ABB RobotStudio station: Path Planning V5 trial.rspag

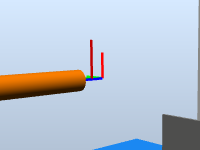
--- station ---
Station Path Planning V5 trial (saved by RobotStudio 6.8.8148.134)
Controller System310, task T_ROB1: task frame (RAPID world) sits at (0, 0, 305) mm in the station
Controller System310
  mechanical unit ROB_1: IRB2600_12_165_C_01, 6 joints, base frame (0, 0, 0) mm
Layout (positions relative to the parent item):
  - Bed [part, from Geometry\Bed.rslib]
  - Nozzle Support [part, from Geometry\Nozzle Support.rslib] at (138.01, 842.67, 817.43) mm, rotated rx -0.73 ry -0.25 rz 45.61 deg
  - Substrate Support [part, from Geometry\Substrate Support.rslib] at (485.68, 958.8, 1236.01) mm, rotated rx -0.25 ry 0.73 rz 135.61 deg
  - Table [part, from Geometry\Table.rslib] at (400.79, 567.93, 822.2) mm, rotated rx -0.73 ry -0.25 rz 45.61 deg
  - IRB2600_12_165_C_01 [mechanism, from Robots\IRB2600_12_165_C_01.rslib] at (0, 0, 305) mm; joint values [1.103, 0.1868, 0.1028, -0.014, 1.2809, 0.3109] (rad or m)
  - substrate_3 [part] at (499.49, 942.27, 926.24) mm, rotated rx -108.89 ry -89.23 rz 154.5 deg
Attachment: Substrate Support is attached to IRB2600_12_165_C_01 / Link6
Attachment: substrate_3 is attached to Substrate Support

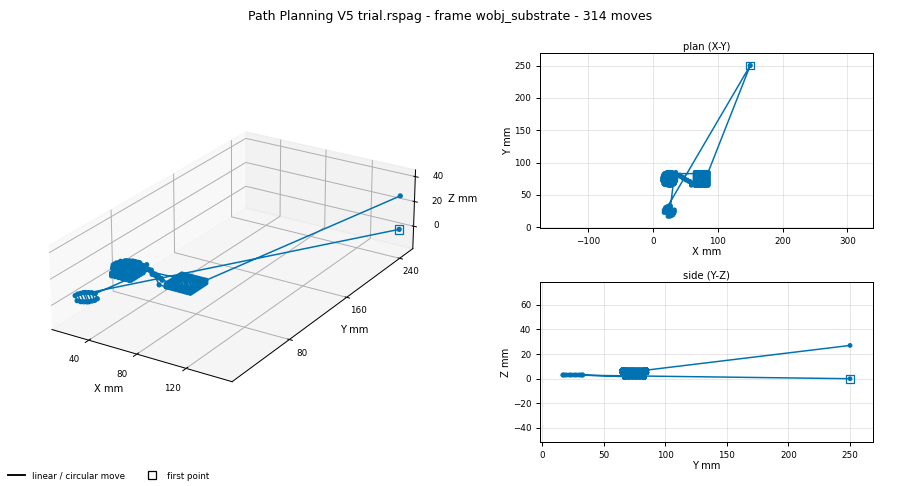
[picture p0: tool path of Path Planning V5 trial.rspag in frame wobj_substrate, 314 of 314 moves have a stored position in this frame; points joined in program order, loops and branches not executed]
--- Backups/System310/RAPID/TASK1/PROGMOD/MainModule.mod ---
MODULE MainModule
    TASK PERS tooldata tool_nozzle:=[FALSE,[[296.65274203,1095.137834363,767.916319098],[0.648657018,0.270531703,-0.654969146,0.277618601]],[1,[0,0,1],[1,0,0,0],0,0,0]];
    TASK PERS wobjdata wobj_substrate:=[TRUE,TRUE,"",[[8.5,-17.5,310],[0.707106781,0,0.707106781,0]],[[0,0,0],[1,0,0,0]]];

    VAR robtarget StartPoint:=[[150,250,0],[1,0,0,0],[-2,0,0,0],[9E+09,9E+09,9E+09,9E+09,9E+09,9E+09]];
    VAR robtarget ReferencePoint:=[[0,0,0],[1,0,0,0],[-2,0,0,0],[9E+09,9E+09,9E+09,9E+09,9E+09,9E+09]];
    VAR speeddata velocity_infill:=[90,500,5000,1000];
    VAR speeddata velocity_edge:=[45,500,5000,1000];
    VAR speeddata velocity_link:=[100,500,5000,1000];
    VAR zonedata zone_infill:=[FALSE,1,1,1,0.1,1,0.1];
    VAR zonedata zone_edge:=[FALSE,0.3,0.3,0.3,0.03,0.3,0.03];
    VAR zonedata zone_link:=[FALSE,5,8,8,0.8,8,0.8];

    PROC main()
        ConfJ\off;
        ConfL\Off;
        WaitTime 1;
        mod20260608;
    ENDPROC

    PROC mod20260608()
        MoveJ StartPoint,v100,fine,tool_nozzle\WObj:=wobj_substrate;
        MoveL RelTool(ReferencePoint,17,23,3\Rx:=0\Ry:=0\Rz:=0),velocity_infill,zone_infill,tool_nozzle\WObj:=wobj_substrate;
        MoveL RelTool(ReferencePoint,23,17,3\Rx:=0\Ry:=0\Rz:=0),velocity_infill,zone_infill,tool_nozzle\WObj:=wobj_substrate;
        MoveL RelTool(ReferencePoint,26,17,3\Rx:=0\Ry:=0\Rz:=0),velocity_infill,zone_infill,tool_nozzle\WObj:=wobj_substrate;
        MoveL RelTool(ReferencePoint,17,26,3\Rx:=0\Ry:=0\Rz:=0),velocity_infill,zone_infill,tool_nozzle\WObj:=wobj_substrate;
        MoveL RelTool(ReferencePoint,18,28,3\Rx:=0\Ry:=0\Rz:=0),velocity_infill,zone_infill,tool_nozzle\WObj:=wobj_substrate;
        MoveL RelTool(ReferencePoint,28,18,3\Rx:=0\Ry:=0\Rz:=0),velocity_infill,zone_infill,tool_nozzle\WObj:=wobj_substrate;
        MoveL RelTool(ReferencePoint,30,19,3\Rx:=0\Ry:=0\Rz:=0),velocity_infill,zone_infill,tool_nozzle\WObj:=wobj_substrate;
        MoveL RelTool(ReferencePoint,19,30,3\Rx:=0\Ry:=0\Rz:=0),velocity_infill,zone_infill,tool_nozzle\WObj:=wobj_substrate;
        MoveL RelTool(ReferencePoint,20,31,3\Rx:=0\Ry:=0\Rz:=0),velocity_infill,zone_infill,tool_nozzle\WObj:=wobj_substrate;
        MoveL RelTool(ReferencePoint,31,20,3\Rx:=0\Ry:=0\Rz:=0),velocity_infill,zone_infill,tool_nozzle\WObj:=wobj_substrate;
        MoveL RelTool(ReferencePoint,32,22,3\Rx:=0\Ry:=0\Rz:=0),velocity_infill,zone_infill,tool_nozzle\WObj:=wobj_substrate;
        MoveL RelTool(ReferencePoint,22,32,3\Rx:=0\Ry:=0\Rz:=0),velocity_infill,zone_infill,tool_nozzle\WObj:=wobj_substrate;
        MoveL RelTool(ReferencePoint,24,33,3\Rx:=0\Ry:=0\Rz:=0),velocity_infill,zone_infill,tool_nozzle\WObj:=wobj_substrate;
        MoveL RelTool(ReferencePoint,33,24,3\Rx:=0\Ry:=0\Rz:=0),velocity_infill,zone_infill,tool_nozzle\WObj:=wobj_substrate;
        MoveL RelTool(ReferencePoint,33,27,3\Rx:=0\Ry:=0\Rz:=0),velocity_infill,zone_infill,tool_nozzle\WObj:=wobj_substrate;
        MoveL RelTool(ReferencePoint,27,33,3\Rx:=0\Ry:=0\Rz:=0),velocity_infill,zone_infill,tool_nozzle\WObj:=wobj_substrate;
        MoveL RelTool(ReferencePoint,33,83,1\Rx:=0\Ry:=0\Rz:=0),velocity_infill,zone_infill,tool_nozzle\WObj:=wobj_substrate;
        MoveL RelTool(ReferencePoint,33,83,1\Rx:=0\Ry:=0\Rz:=0),velocity_infill,zone_infill,tool_nozzle\WObj:=wobj_substrate;
        MoveL RelTool(ReferencePoint,33,80,1\Rx:=0\Ry:=0\Rz:=0),velocity_infill,zone_infill,tool_nozzle\WObj:=wobj_substrate;
        MoveL RelTool(ReferencePoint,30,83,1\Rx:=0\Ry:=0\Rz:=0),velocity_infill,zone_infill,tool_nozzle\WObj:=wobj_substrate;
        MoveL RelTool(ReferencePoint,27,83,1\Rx:=0\Ry:=0\Rz:=0),velocity_infill,zone_infill,tool_nozzle\WObj:=wobj_substrate;
        MoveL RelTool(ReferencePoint,33,77,1\Rx:=0\Ry:=0\Rz:=0),velocity_infill,zone_infill,tool_nozzle\WObj:=wobj_substrate;
        MoveL RelTool(ReferencePoint,33,74,1\Rx:=0\Ry:=0\Rz:=0),velocity_infill,zone_infill,tool_nozzle\WObj:=wobj_substrate;
        MoveL RelTool(ReferencePoint,24,83,1\Rx:=0\Ry:=0\Rz:=0),velocity_infill,zone_infill,tool_nozzle\WObj:=wobj_substrate;
        MoveL RelTool(ReferencePoint,21,83,1\Rx:=0\Ry:=0\Rz:=0),velocity_infill,zone_infill,tool_nozzle\WObj:=wobj_substrate;
        MoveL RelTool(ReferencePoint,33,71,1\Rx:=0\Ry:=0\Rz:=0),velocity_infill,zone_infill,tool_nozzle\WObj:=wobj_substrate;
        MoveL RelTool(ReferencePoint,33,68,1\Rx:=0\Ry:=0\Rz:=0),velocity_infill,zone_infill,tool_nozzle\WObj:=wobj_substrate;
        MoveL RelTool(ReferencePoint,18,83,1\Rx:=0\Ry:=0\Rz:=0),velocity_infill,zone_infill,tool_nozzle\WObj:=wobj_substrate;
        MoveL RelTool(ReferencePoint,17,82,1\Rx:=0\Ry:=0\Rz:=0),velocity_infill,zone_infill,tool_nozzle\WObj:=wobj_substrate;
        MoveL RelTool(ReferencePoint,32,67,1\Rx:=0\Ry:=0\Rz:=0),velocity_infill,zone_infill,tool_nozzle\WObj:=wobj_substrate;
        MoveL RelTool(ReferencePoint,29,67,1\Rx:=0\Ry:=0\Rz:=0),velocity_infill,zone_infill,tool_nozzle\WObj:=wobj_substrate;
        MoveL RelTool(ReferencePoint,17,79,1\Rx:=0\Ry:=0\Rz:=0),velocity_infill,zone_infill,tool_nozzle\WObj:=wobj_substrate;
        MoveL RelTool(ReferencePoint,17,76,1\Rx:=0\Ry:=0\Rz:=0),velocity_infill,zone_infill,tool_nozzle\WObj:=wobj_substrate;
        MoveL RelTool(ReferencePoint,26,67,1\Rx:=0\Ry:=0\Rz:=0),velocity_infill,zone_infill,tool_nozzle\WObj:=wobj_substrate;
        MoveL RelTool(ReferencePoint,23,67,1\Rx:=0\Ry:=0\Rz:=0),velocity_infill,zone_infill,tool_nozzle\WObj:=wobj_substrate;
        MoveL RelTool(ReferencePoint,17,73,1\Rx:=0\Ry:=0\Rz:=0),velocity_infill,zone_infill,tool_nozzle\WObj:=wobj_substrate;
        MoveL RelTool(ReferencePoint,17,70,1\Rx:=0\Ry:=0\Rz:=0),velocity_infill,zone_infill,tool_nozzle\WObj:=wobj_substrate;
        MoveL RelTool(ReferencePoint,20,67,1\Rx:=0\Ry:=0\Rz:=0),velocity_infill,zone_infill,tool_nozzle\WObj:=wobj_substrate;
        MoveL RelTool(ReferencePoint,17,67,1\Rx:=0\Ry:=0\Rz:=0),velocity_infill,zone_infill,tool_nozzle\WObj:=wobj_substrate;
        MoveL RelTool(ReferencePoint,17,67,1\Rx:=0\Ry:=0\Rz:=0),velocity_infill,zone_infill,tool_nozzle\WObj:=wobj_substrate;
        MoveL RelTool(ReferencePoint,17,67,3\Rx:=0\Ry:=0\Rz:=0),velocity_infill,zone_infill,tool_nozzle\WObj:=wobj_substrate;
        MoveL RelTool(ReferencePoint,17,67,3\Rx:=0\Ry:=0\Rz:=0),velocity_infill,zone_infill,tool_nozzle\WObj:=wobj_substrate;
        MoveL RelTool(ReferencePoint,20,67,3\Rx:=0\Ry:=0\Rz:=0),velocity_infill,zone_infill,tool_nozzle\WObj:=wobj_substrate;
        MoveL RelTool(ReferencePoint,17,70,3\Rx:=0\Ry:=0\Rz:=0),velocity_infill,zone_infill,tool_nozzle\WObj:=wobj_substrate;
        MoveL RelTool(ReferencePoint,17,73,3\Rx:=0\Ry:=0\Rz:=0),velocity_infill,zone_infill,tool_nozzle\WObj:=wobj_substrate;
        MoveL RelTool(ReferencePoint,23,67,3\Rx:=0\Ry:=0\Rz:=0),velocity_infill,zone_infill,tool_nozzle\WObj:=wobj_substrate;
        MoveL RelTool(ReferencePoint,26,67,3\Rx:=0\Ry:=0\Rz:=0),velocity_infill,zone_infill,tool_nozzle\WObj:=wobj_substrate;
        MoveL RelTool(ReferencePoint,17,76,3\Rx:=0\Ry:=0\Rz:=0),velocity_infill,zone_infill,tool_nozzle\WObj:=wobj_substrate;
        MoveL RelTool(ReferencePoint,17,79,3\Rx:=0\Ry:=0\Rz:=0),velocity_infill,zone_infill,tool_nozzle\WObj:=wobj_substrate;
        MoveL RelTool(ReferencePoint,29,67,3\Rx:=0\Ry:=0\Rz:=0),velocity_infill,zone_infill,tool_nozzle\WObj:=wobj_substrate;
        MoveL RelTool(ReferencePoint,32,67,3\Rx:=0\Ry:=0\Rz:=0),velocity_infill,zone_infill,tool_nozzle\WObj:=wobj_substrate;
        MoveL RelTool(ReferencePoint,17,82,3\Rx:=0\Ry:=0\Rz:=0),velocity_infill,zone_infill,tool_nozzle\WObj:=wobj_substrate;
        MoveL RelTool(ReferencePoint,18,83,3\Rx:=0\Ry:=0\Rz:=0),velocity_infill,zone_infill,tool_nozzle\WObj:=wobj_substrate;
        MoveL RelTool(ReferencePoint,33,68,3\Rx:=0\Ry:=0\Rz:=0),velocity_infill,zone_infill,tool_nozzle\WObj:=wobj_substrate;
        MoveL RelTool(ReferencePoint,33,71,3\Rx:=0\Ry:=0\Rz:=0),velocity_infill,zone_infill,tool_nozzle\WObj:=wobj_substrate;
        MoveL RelTool(ReferencePoint,21,83,3\Rx:=0\Ry:=0\Rz:=0),velocity_infill,zone_infill,tool_nozzle\WObj:=wobj_substrate;
        MoveL RelTool(ReferencePoint,24,83,3\Rx:=0\Ry:=0\Rz:=0),velocity_infill,zone_infill,tool_nozzle\WObj:=wobj_substrate;
        MoveL RelTool(ReferencePoint,33,74,3\Rx:=0\Ry:=0\Rz:=0),velocity_infill,zone_infill,tool_nozzle\WObj:=wobj_substrate;
        MoveL RelTool(ReferencePoint,33,77,3\Rx:=0\Ry:=0\Rz:=0),velocity_infill,zone_infill,tool_nozzle\WObj:=wobj_substrate;
        MoveL RelTool(ReferencePoint,27,83,3\Rx:=0\Ry:=0\Rz:=0),velocity_infill,zone_infill,tool_nozzle\WObj:=wobj_substrate;
        MoveL RelTool(ReferencePoint,30,83,3\Rx:=0\Ry:=0\Rz:=0),velocity_infill,zone_infill,tool_nozzle\WObj:=wobj_substrate;
        MoveL RelTool(ReferencePoint,33,80,3\Rx:=0\Ry:=0\Rz:=0),velocity_infill,zone_infill,tool_nozzle\WObj:=wobj_substrate;
        MoveL RelTool(ReferencePoint,33,83,3\Rx:=0\Ry:=0\Rz:=0),velocity_infill,zone_infill,tool_nozzle\WObj:=wobj_substrate;
        MoveL RelTool(ReferencePoint,33,83,3\Rx:=0\Ry:=0\Rz:=0),velocity_infill,zone_infill,tool_nozzle\WObj:=wobj_substrate;
        MoveL RelTool(ReferencePoint,83,83,5\Rx:=0\Ry:=0\Rz:=0),velocity_infill,zone_infill,tool_nozzle\WObj:=wobj_substrate;
        MoveL RelTool(ReferencePoint,83,83,5\Rx:=0\Ry:=0\Rz:=0),velocity_infill,zone_infill,tool_nozzle\WObj:=wobj_substrate;
        MoveL RelTool(ReferencePoint,83,80,5\Rx:=0\Ry:=0\Rz:=0),velocity_infill,zone_infill,tool_nozzle\WObj:=wobj_substrate;
        MoveL RelTool(ReferencePoint,80,83,5\Rx:=0\Ry:=0\Rz:=0),velocity_infill,zone_infill,tool_nozzle\WObj:=wobj_substrate;
        MoveL RelTool(ReferencePoint,77,83,5\Rx:=0\Ry:=0\Rz:=0),velocity_infill,zone_infill,tool_nozzle\WObj:=wobj_substrate;
        MoveL RelTool(ReferencePoint,83,77,5\Rx:=0\Ry:=0\Rz:=0),velocity_infill,zone_infill,tool_nozzle\WObj:=wobj_substrate;
        MoveL RelTool(ReferencePoint,83,74,5\Rx:=0\Ry:=0\Rz:=0),velocity_infill,zone_infill,tool_nozzle\WObj:=wobj_substrate;
        MoveL RelTool(ReferencePoint,74,83,5\Rx:=0\Ry:=0\Rz:=0),velocity_infill,zone_infill,tool_nozzle\WObj:=wobj_substrate;
        MoveL RelTool(ReferencePoint,71,83,5\Rx:=0\Ry:=0\Rz:=0),velocity_infill,zone_infill,tool_nozzle\WObj:=wobj_substrate;
        MoveL RelTool(ReferencePoint,83,71,5\Rx:=0\Ry:=0\Rz:=0),velocity_infill,zone_infill,tool_nozzle\WObj:=wobj_substrate;
        MoveL RelTool(ReferencePoint,83,68,5\Rx:=0\Ry:=0\Rz:=0),velocity_infill,zone_infill,tool_nozzle\WObj:=wobj_substrate;
        MoveL RelTool(ReferencePoint,68,83,5\Rx:=0\Ry:=0\Rz:=0),velocity_infill,zone_infill,tool_nozzle\WObj:=wobj_substrate;
        MoveL RelTool(ReferencePoint,67,82,5\Rx:=0\Ry:=0\Rz:=0),velocity_infill,zone_infill,tool_nozzle\WObj:=wobj_substrate;
        MoveL RelTool(ReferencePoint,82,67,5\Rx:=0\Ry:=0\Rz:=0),velocity_infill,zone_infill,tool_nozzle\WObj:=wobj_substrate;
        MoveL RelTool(ReferencePoint,79,67,5\Rx:=0\Ry:=0\Rz:=0),velocity_infill,zone_infill,tool_nozzle\WObj:=wobj_substrate;
        MoveL RelTool(ReferencePoint,67,79,5\Rx:=0\Ry:=0\Rz:=0),velocity_infill,zone_infill,tool_nozzle\WObj:=wobj_substrate;
        MoveL RelTool(ReferencePoint,67,76,5\Rx:=0\Ry:=0\Rz:=0),velocity_infill,zone_infill,tool_nozzle\WObj:=wobj_substrate;
        MoveL RelTool(ReferencePoint,76,67,5\Rx:=0\Ry:=0\Rz:=0),velocity_infill,zone_infill,tool_nozzle\WObj:=wobj_substrate;
        MoveL RelTool(ReferencePoint,73,67,5\Rx:=0\Ry:=0\Rz:=0),velocity_infill,zone_infill,tool_nozzle\WObj:=wobj_substrate;
        MoveL RelTool(ReferencePoint,67,73,5\Rx:=0\Ry:=0\Rz:=0),velocity_infill,zone_infill,tool_nozzle\WObj:=wobj_substrate;
        MoveL RelTool(ReferencePoint,67,70,5\Rx:=0\Ry:=0\Rz:=0),velocity_infill,zone_infill,tool_nozzle\WObj:=wobj_substrate;
        MoveL RelTool(ReferencePoint,70,67,5\Rx:=0\Ry:=0\Rz:=0),velocity_infill,zone_infill,tool_nozzle\WObj:=wobj_substrate;
        MoveL RelTool(ReferencePoint,67,67,5\Rx:=0\Ry:=0\Rz:=0),velocity_infill,zone_infill,tool_nozzle\WObj:=wobj_substrate;
        MoveL RelTool(ReferencePoint,67,67,5\Rx:=0\Ry:=0\Rz:=0),velocity_infill,zone_infill,tool_nozzle\WObj:=wobj_substrate;
        MoveL RelTool(ReferencePoint,65,65,5\Rx:=0\Ry:=-30\Rz:=0),velocity_edge,zone_edge,tool_nozzle\WObj:=wobj_substrate;
        MoveL RelTool(ReferencePoint,65,67,5\Rx:=0\Ry:=-30\Rz:=0),velocity_edge,zone_edge,tool_nozzle\WObj:=wobj_substrate;
        MoveL RelTool(ReferencePoint,65,69,5\Rx:=0\Ry:=-30\Rz:=0),velocity_edge,zone_edge,tool_nozzle\WObj:=wobj_substrate;
        MoveL RelTool(ReferencePoint,65,71,5\Rx:=0\Ry:=-30\Rz:=0),velocity_edge,zone_edge,tool_nozzle\WObj:=wobj_substrate;
        MoveL RelTool(ReferencePoint,65,73,5\Rx:=0\Ry:=-30\Rz:=0),velocity_edge,zone_edge,tool_nozzle\WObj:=wobj_substrate;
        MoveL RelTool(ReferencePoint,65,75,5\Rx:=0\Ry:=-30\Rz:=0),velocity_edge,zone_edge,tool_nozzle\WObj:=wobj_substrate;
        MoveL RelTool(ReferencePoint,65,77,5\Rx:=0\Ry:=-30\Rz:=0),velocity_edge,zone_edge,tool_nozzle\WObj:=wobj_substrate;
        MoveL RelTool(ReferencePoint,65,79,5\Rx:=0\Ry:=-30\Rz:=0),velocity_edge,zone_edge,tool_nozzle\WObj:=wobj_substrate;
        MoveL RelTool(ReferencePoint,65,81,5\Rx:=0\Ry:=-30\Rz:=0),velocity_edge,zone_edge,tool_nozzle\WObj:=wobj_substrate;
        MoveL RelTool(ReferencePoint,65,83,5\Rx:=0\Ry:=-30\Rz:=0),velocity_edge,zone_edge,tool_nozzle\WObj:=wobj_substrate;
        MoveL RelTool(ReferencePoint,65,85,5\Rx:=-30\Ry:=0\Rz:=0),velocity_edge,zone_edge,tool_nozzle\WObj:=wobj_substrate;
        MoveL RelTool(ReferencePoint,67,85,5\Rx:=-30\Ry:=0\Rz:=0),velocity_edge,zone_edge,tool_nozzle\WObj:=wobj_substrate;
        MoveL RelTool(ReferencePoint,69,85,5\Rx:=-30\Ry:=0\Rz:=0),velocity_edge,zone_edge,tool_nozzle\WObj:=wobj_substrate;
        MoveL RelTool(ReferencePoint,71,85,5\Rx:=-30\Ry:=0\Rz:=0),velocity_edge,zone_edge,tool_nozzle\WObj:=wobj_substrate;
        MoveL RelTool(ReferencePoint,73,85,5\Rx:=-30\Ry:=0\Rz:=0),velocity_edge,zone_edge,tool_nozzle\WObj:=wobj_substrate;
        MoveL RelTool(ReferencePoint,75,85,5\Rx:=-30\Ry:=0\Rz:=0),velocity_edge,zone_edge,tool_nozzle\WObj:=wobj_substrate;
        MoveL RelTool(ReferencePoint,77,85,5\Rx:=-30\Ry:=0\Rz:=0),velocity_edge,zone_edge,tool_nozzle\WObj:=wobj_substrate;
        MoveL RelTool(ReferencePoint,79,85,5\Rx:=-30\Ry:=0\Rz:=0),velocity_edge,zone_edge,tool_nozzle\WObj:=wobj_substrate;
        MoveL RelTool(ReferencePoint,81,85,5\Rx:=-30\Ry:=0\Rz:=0),velocity_edge,zone_edge,tool_nozzle\WObj:=wobj_substrate;
        MoveL RelTool(ReferencePoint,83,85,5\Rx:=-30\Ry:=0\Rz:=0),velocity_edge,zone_edge,tool_nozzle\WObj:=wobj_substrate;
        MoveL RelTool(ReferencePoint,85,85,5\Rx:=0\Ry:=30\Rz:=0),velocity_edge,zone_edge,tool_nozzle\WObj:=wobj_substrate;
        MoveL RelTool(ReferencePoint,85,83,5\Rx:=0\Ry:=30\Rz:=0),velocity_edge,zone_edge,tool_nozzle\WObj:=wobj_substrate;
        MoveL RelTool(ReferencePoint,85,81,5\Rx:=0\Ry:=30\Rz:=0),velocity_edge,zone_edge,tool_nozzle\WObj:=wobj_substrate;
        MoveL RelTool(ReferencePoint,85,79,5\Rx:=0\Ry:=30\Rz:=0),velocity_edge,zone_edge,tool_nozzle\WObj:=wobj_substrate;
        MoveL RelTool(ReferencePoint,85,77,5\Rx:=0\Ry:=30\Rz:=0),velocity_edge,zone_edge,tool_nozzle\WObj:=wobj_substrate;
        MoveL RelTool(ReferencePoint,85,75,5\Rx:=0\Ry:=30\Rz:=0),velocity_edge,zone_edge,tool_nozzle\WObj:=wobj_substrate;
        MoveL RelTool(ReferencePoint,85,73,5\Rx:=0\Ry:=30\Rz:=0),velocity_edge,zone_edge,tool_nozzle\WObj:=wobj_substrate;
        MoveL RelTool(ReferencePoint,85,71,5\Rx:=0\Ry:=30\Rz:=0),velocity_edge,zone_edge,tool_nozzle\WObj:=wobj_substrate;
        MoveL RelTool(ReferencePoint,85,69,5\Rx:=0\Ry:=30\Rz:=0),velocity_edge,zone_edge,tool_nozzle\WObj:=wobj_substrate;
        MoveL RelTool(ReferencePoint,85,67,5\Rx:=0\Ry:=30\Rz:=0),velocity_edge,zone_edge,tool_nozzle\WObj:=wobj_substrate;
        MoveL RelTool(ReferencePoint,85,65,5\Rx:=30\Ry:=0\Rz:=0),velocity_edge,zone_edge,tool_nozzle\WObj:=wobj_substrate;
        MoveL RelTool(ReferencePoint,83,65,5\Rx:=30\Ry:=0\Rz:=0),velocity_edge,zone_edge,tool_nozzle\WObj:=wobj_substrate;
        MoveL RelTool(ReferencePoint,81,65,5\Rx:=30\Ry:=0\Rz:=0),velocity_edge,zone_edge,tool_nozzle\WObj:=wobj_substrate;
        MoveL RelTool(ReferencePoint,79,65,5\Rx:=30\Ry:=0\Rz:=0),velocity_edge,zone_edge,tool_nozzle\WObj:=wobj_substrate;
        MoveL RelTool(ReferencePoint,77,65,5\Rx:=30\Ry:=0\Rz:=0),velocity_edge,zone_edge,tool_nozzle\WObj:=wobj_substrate;
        MoveL RelTool(ReferencePoint,75,65,5\Rx:=30\Ry:=0\Rz:=0),velocity_edge,zone_edge,tool_nozzle\WObj:=wobj_substrate;
        MoveL RelTool(ReferencePoint,73,65,5\Rx:=30\Ry:=0\Rz:=0),velocity_edge,zone_edge,tool_nozzle\WObj:=wobj_substrate;
        MoveL RelTool(ReferencePoint,71,65,5\Rx:=30\Ry:=0\Rz:=0),velocity_edge,zone_edge,tool_nozzle\WObj:=wobj_substrate;
        MoveL RelTool(ReferencePoint,69,65,5\Rx:=30\Ry:=0\Rz:=0),velocity_edge,zone_edge,tool_nozzle\WObj:=wobj_substrate;
        MoveL RelTool(ReferencePoint,67,65,5\Rx:=30\Ry:=0\Rz:=0),velocity_edge,zone_edge,tool_nozzle\WObj:=wobj_substrate;
        MoveL RelTool(ReferencePoint,65,65,5\Rx:=30\Ry:=0\Rz:=0),velocity_edge,zone_edge,tool_nozzle\WObj:=wobj_substrate;
        MoveL RelTool(ReferencePoint,65,65,5\Rx:=0\Ry:=0\Rz:=0),velocity_link,zone_link,tool_nozzle\WObj:=wobj_substrate;
        MoveL RelTool(ReferencePoint,59,65,5\Rx:=0\Ry:=0\Rz:=0),velocity_link,zone_link,tool_nozzle\WObj:=wobj_substrate;
        MoveL RelTool(ReferencePoint,47,77,5\Rx:=0\Ry:=0\Rz:=0),velocity_link,zone_link,tool_nozzle\WObj:=wobj_substrate;
        MoveL RelTool(ReferencePoint,45,77,5\Rx:=0\Ry:=0\Rz:=0),velocity_link,zone_link,tool_nozzle\WObj:=wobj_substrate;
        MoveL RelTool(ReferencePoint,41,81,5\Rx:=0\Ry:=0\Rz:=0),velocity_link,zone_link,tool_nozzle\WObj:=wobj_substrate;
        MoveL RelTool(ReferencePoint,37,81,5\Rx:=0\Ry:=0\Rz:=0),velocity_link,zone_link,tool_nozzle\WObj:=wobj_substrate;
        MoveL RelTool(ReferencePoint,35,83,5\Rx:=0\Ry:=0\Rz:=0),velocity_link,zone_link,tool_nozzle\WObj:=wobj_substrate;
        MoveL RelTool(ReferencePoint,29,83,5\Rx:=0\Ry:=0\Rz:=0),velocity_link,zone_link,tool_nozzle\WObj:=wobj_substrate;
        MoveL RelTool(ReferencePoint,27,83,5\Rx:=0\Ry:=0\Rz:=0),velocity_infill,zone_infill,tool_nozzle\WObj:=wobj_substrate;
        MoveL RelTool(ReferencePoint,33,77,5\Rx:=0\Ry:=0\Rz:=0),velocity_infill,zone_infill,tool_nozzle\WObj:=wobj_substrate;
        MoveL RelTool(ReferencePoint,33,74,5\Rx:=0\Ry:=0\Rz:=0),velocity_infill,zone_infill,tool_nozzle\WObj:=wobj_substrate;
        MoveL RelTool(ReferencePoint,24,83,5\Rx:=0\Ry:=0\Rz:=0),velocity_infill,zone_infill,tool_nozzle\WObj:=wobj_substrate;
        MoveL RelTool(ReferencePoint,22,82,5\Rx:=0\Ry:=0\Rz:=0),velocity_infill,zone_infill,tool_nozzle\WObj:=wobj_substrate;
        MoveL RelTool(ReferencePoint,32,72,5\Rx:=0\Ry:=0\Rz:=0),velocity_infill,zone_infill,tool_nozzle\WObj:=wobj_substrate;
        MoveL RelTool(ReferencePoint,31,70,5\Rx:=0\Ry:=0\Rz:=0),velocity_infill,zone_infill,tool_nozzle\WObj:=wobj_substrate;
        MoveL RelTool(ReferencePoint,20,81,5\Rx:=0\Ry:=0\Rz:=0),velocity_infill,zone_infill,tool_nozzle\WObj:=wobj_substrate;
        MoveL RelTool(ReferencePoint,19,80,5\Rx:=0\Ry:=0\Rz:=0),velocity_infill,zone_infill,tool_nozzle\WObj:=wobj_substrate;
        MoveL RelTool(ReferencePoint,30,69,5\Rx:=0\Ry:=0\Rz:=0),velocity_infill,zone_infill,tool_nozzle\WObj:=wobj_substrate;
        MoveL RelTool(ReferencePoint,28,68,5\Rx:=0\Ry:=0\Rz:=0),velocity_infill,zone_infill,tool_nozzle\WObj:=wobj_substrate;
        MoveL RelTool(ReferencePoint,18,78,5\Rx:=0\Ry:=0\Rz:=0),velocity_infill,zone_infill,tool_nozzle\WObj:=wobj_substrate;
        MoveL RelTool(ReferencePoint,17,76,5\Rx:=0\Ry:=0\Rz:=0),velocity_infill,zone_infill,tool_nozzle\WObj:=wobj_substrate;
        MoveL RelTool(ReferencePoint,26,67,5\Rx:=0\Ry:=0\Rz:=0),velocity_infill,zone_infill,tool_nozzle\WObj:=wobj_substrate;
        MoveL RelTool(ReferencePoint,23,67,5\Rx:=0\Ry:=0\Rz:=0),velocity_infill,zone_infill,tool_nozzle\WObj:=wobj_substrate;
        MoveL RelTool(ReferencePoint,17,73,5\Rx:=0\Ry:=0\Rz:=0),velocity_infill,zone_infill,tool_nozzle\WObj:=wobj_substrate;
        MoveL RelTool(ReferencePoint,15,72,5\Rx:=8\Ry:=-29\Rz:=0),velocity_edge,zone_edge,tool_nozzle\WObj:=wobj_substrate;
        MoveL RelTool(ReferencePoint,15,74,5\Rx:=2\Ry:=-30\Rz:=0),velocity_edge,zone_edge,tool_nozzle\WObj:=wobj_substrate;
        MoveL RelTool(ReferencePoint,15,76,5\Rx:=-5\Ry:=-30\Rz:=0),velocity_edge,zone_edge,tool_nozzle\WObj:=wobj_substrate;
        MoveL RelTool(ReferencePoint,15,78,5\Rx:=-11\Ry:=-28\Rz:=0),velocity_edge,zone_edge,tool_nozzle\WObj:=wobj_substrate;
        MoveL RelTool(ReferencePoint,16,80,5\Rx:=-17\Ry:=-25\Rz:=0),velocity_edge,zone_edge,tool_nozzle\WObj:=wobj_substrate;
        MoveL RelTool(ReferencePoint,17,81,5\Rx:=-21\Ry:=-22\Rz:=0),velocity_edge,zone_edge,tool_nozzle\WObj:=wobj_substrate;
        MoveL RelTool(ReferencePoint,19,83,5\Rx:=-25\Ry:=-17\Rz:=0),velocity_edge,zone_edge,tool_nozzle\WObj:=wobj_substrate;
        MoveL RelTool(ReferencePoint,21,84,5\Rx:=-28\Ry:=-12\Rz:=0),velocity_edge,zone_edge,tool_nozzle\WObj:=wobj_substrate;
        MoveL RelTool(ReferencePoint,22,85,5\Rx:=-29\Ry:=-7\Rz:=0),velocity_edge,zone_edge,tool_nozzle\WObj:=wobj_substrate;
        MoveL RelTool(ReferencePoint,24,85,5\Rx:=-30\Ry:=-1\Rz:=0),velocity_edge,zone_edge,tool_nozzle\WObj:=wobj_substrate;
        MoveL RelTool(ReferencePoint,26,85,5\Rx:=-30\Ry:=4\Rz:=0),velocity_edge,zone_edge,tool_nozzle\WObj:=wobj_substrate;
        MoveL RelTool(ReferencePoint,28,84,5\Rx:=-29\Ry:=10\Rz:=0),velocity_edge,zone_edge,tool_nozzle\WObj:=wobj_substrate;
        MoveL RelTool(ReferencePoint,30,84,5\Rx:=-26\Ry:=15\Rz:=0),velocity_edge,zone_edge,tool_nozzle\WObj:=wobj_substrate;
        MoveL RelTool(ReferencePoint,32,82,5\Rx:=-23\Ry:=20\Rz:=0),velocity_edge,zone_edge,tool_nozzle\WObj:=wobj_substrate;
        MoveL RelTool(ReferencePoint,33,81,5\Rx:=-19\Ry:=24\Rz:=0),velocity_edge,zone_edge,tool_nozzle\WObj:=wobj_substrate;
        MoveL RelTool(ReferencePoint,34,79,5\Rx:=-14\Ry:=27\Rz:=0),velocity_edge,zone_edge,tool_nozzle\WObj:=wobj_substrate;
        MoveL RelTool(ReferencePoint,35,77,5\Rx:=-8\Ry:=29\Rz:=0),velocity_edge,zone_edge,tool_nozzle\WObj:=wobj_substrate;
        MoveL RelTool(ReferencePoint,35,75,5\Rx:=-2\Ry:=30\Rz:=0),velocity_edge,zone_edge,tool_nozzle\WObj:=wobj_substrate;
        MoveL RelTool(ReferencePoint,35,73,5\Rx:=5\Ry:=30\Rz:=0),velocity_edge,zone_edge,tool_nozzle\WObj:=wobj_substrate;
        MoveL RelTool(ReferencePoint,34,71,5\Rx:=11\Ry:=28\Rz:=0),velocity_edge,zone_edge,tool_nozzle\WObj:=wobj_substrate;
        MoveL RelTool(ReferencePoint,33,70,5\Rx:=17\Ry:=25\Rz:=0),velocity_edge,zone_edge,tool_nozzle\WObj:=wobj_substrate;
        MoveL RelTool(ReferencePoint,32,68,5\Rx:=21\Ry:=22\Rz:=0),velocity_edge,zone_edge,tool_nozzle\WObj:=wobj_substrate;
        MoveL RelTool(ReferencePoint,31,67,5\Rx:=25\Ry:=17\Rz:=0),velocity_edge,zone_edge,tool_nozzle\WObj:=wobj_substrate;
        MoveL RelTool(ReferencePoint,29,66,5\Rx:=28\Ry:=12\Rz:=0),velocity_edge,zone_edge,tool_nozzle\WObj:=wobj_substrate;
        MoveL RelTool(ReferencePoint,27,65,5\Rx:=29\Ry:=7\Rz:=0),velocity_edge,zone_edge,tool_nozzle\WObj:=wobj_substrate;
        MoveL RelTool(ReferencePoint,25,65,5\Rx:=30\Ry:=1\Rz:=0),velocity_edge,zone_edge,tool_nozzle\WObj:=wobj_substrate;
        MoveL RelTool(ReferencePoint,23,65,5\Rx:=30\Ry:=-4\Rz:=0),velocity_edge,zone_edge,tool_nozzle\WObj:=wobj_substrate;
        MoveL RelTool(ReferencePoint,21,66,5\Rx:=28\Ry:=-12\Rz:=0),velocity_edge,zone_edge,tool_nozzle\WObj:=wobj_substrate;
        MoveL RelTool(ReferencePoint,19,67,5\Rx:=25\Ry:=-17\Rz:=0),velocity_edge,zone_edge,tool_nozzle\WObj:=wobj_substrate;
        MoveL RelTool(ReferencePoint,18,68,5\Rx:=21\Ry:=-22\Rz:=0),velocity_edge,zone_edge,tool_nozzle\WObj:=wobj_substrate;
        MoveL RelTool(ReferencePoint,17,70,5\Rx:=17\Ry:=-25\Rz:=0),velocity_edge,zone_edge,tool_nozzle\WObj:=wobj_substrate;
        MoveL RelTool(ReferencePoint,16,71,5\Rx:=11\Ry:=-28\Rz:=0),velocity_edge,zone_edge,tool_nozzle\WObj:=wobj_substrate;
        MoveL RelTool(ReferencePoint,15,72,5\Rx:=9\Ry:=-29\Rz:=0),velocity_edge,zone_edge,tool_nozzle\WObj:=wobj_substrate;
        MoveL RelTool(ReferencePoint,17,73,7\Rx:=0\Ry:=0\Rz:=0),velocity_infill,zone_infill,tool_nozzle\WObj:=wobj_substrate;
        MoveL RelTool(ReferencePoint,23,67,7\Rx:=0\Ry:=0\Rz:=0),velocity_infill,zone_infill,tool_nozzle\WObj:=wobj_substrate;
        MoveL RelTool(ReferencePoint,26,67,7\Rx:=0\Ry:=0\Rz:=0),velocity_infill,zone_infill,tool_nozzle\WObj:=wobj_substrate;
        MoveL RelTool(ReferencePoint,17,76,7\Rx:=0\Ry:=0\Rz:=0),velocity_infill,zone_infill,tool_nozzle\WObj:=wobj_substrate;
        MoveL RelTool(ReferencePoint,18,78,7\Rx:=0\Ry:=0\Rz:=0),velocity_infill,zone_infill,tool_nozzle\WObj:=wobj_substrate;
        MoveL RelTool(ReferencePoint,28,68,7\Rx:=0\Ry:=0\Rz:=0),velocity_infill,zone_infill,tool_nozzle\WObj:=wobj_substrate;
        MoveL RelTool(ReferencePoint,30,69,7\Rx:=0\Ry:=0\Rz:=0),velocity_infill,zone_infill,tool_nozzle\WObj:=wobj_substrate;
        MoveL RelTool(ReferencePoint,19,80,7\Rx:=0\Ry:=0\Rz:=0),velocity_infill,zone_infill,tool_nozzle\WObj:=wobj_substrate;
        MoveL RelTool(ReferencePoint,20,81,7\Rx:=0\Ry:=0\Rz:=0),velocity_infill,zone_infill,tool_nozzle\WObj:=wobj_substrate;
        MoveL RelTool(ReferencePoint,31,70,7\Rx:=0\Ry:=0\Rz:=0),velocity_infill,zone_infill,tool_nozzle\WObj:=wobj_substrate;
        MoveL RelTool(ReferencePoint,32,72,7\Rx:=0\Ry:=0\Rz:=0),velocity_infill,zone_infill,tool_nozzle\WObj:=wobj_substrate;
        MoveL RelTool(ReferencePoint,22,82,7\Rx:=0\Ry:=0\Rz:=0),velocity_infill,zone_infill,tool_nozzle\WObj:=wobj_substrate;
        MoveL RelTool(ReferencePoint,24,83,7\Rx:=0\Ry:=0\Rz:=0),velocity_infill,zone_infill,tool_nozzle\WObj:=wobj_substrate;
        MoveL RelTool(ReferencePoint,33,74,7\Rx:=0\Ry:=0\Rz:=0),velocity_infill,zone_infill,tool_nozzle\WObj:=wobj_substrate;
        MoveL RelTool(ReferencePoint,33,77,7\Rx:=0\Ry:=0\Rz:=0),velocity_infill,zone_infill,tool_nozzle\WObj:=wobj_substrate;
        MoveL RelTool(ReferencePoint,27,83,7\Rx:=0\Ry:=0\Rz:=0),velocity_infill,zone_infill,tool_nozzle\WObj:=wobj_substrate;
        MoveL RelTool(ReferencePoint,28,85,7\Rx:=-29\Ry:=7\Rz:=0),velocity_edge,zone_edge,tool_nozzle\WObj:=wobj_substrate;
        MoveL RelTool(ReferencePoint,29,84,7\Rx:=-28\Ry:=12\Rz:=0),velocity_edge,zone_edge,tool_nozzle\WObj:=wobj_substrate;
        MoveL RelTool(ReferencePoint,31,83,7\Rx:=-24\Ry:=18\Rz:=0),velocity_edge,zone_edge,tool_nozzle\WObj:=wobj_substrate;
        MoveL RelTool(ReferencePoint,33,82,7\Rx:=-21\Ry:=22\Rz:=0),velocity_edge,zone_edge,tool_nozzle\WObj:=wobj_substrate;
        MoveL RelTool(ReferencePoint,34,80,7\Rx:=-15\Ry:=26\Rz:=0),velocity_edge,zone_edge,tool_nozzle\WObj:=wobj_substrate;
        MoveL RelTool(ReferencePoint,34,78,7\Rx:=-11\Ry:=28\Rz:=0),velocity_edge,zone_edge,tool_nozzle\WObj:=wobj_substrate;
        MoveL RelTool(ReferencePoint,35,76,7\Rx:=-2\Ry:=30\Rz:=0),velocity_edge,zone_edge,tool_nozzle\WObj:=wobj_substrate;
        MoveL RelTool(ReferencePoint,35,74,7\Rx:=2\Ry:=30\Rz:=0),velocity_edge,zone_edge,tool_nozzle\WObj:=wobj_substrate;
        MoveL RelTool(ReferencePoint,35,72,7\Rx:=8\Ry:=29\Rz:=0),velocity_edge,zone_edge,tool_nozzle\WObj:=wobj_substrate;
        MoveL RelTool(ReferencePoint,34,70,7\Rx:=15\Ry:=26\Rz:=0),velocity_edge,zone_edge,tool_nozzle\WObj:=wobj_substrate;
        MoveL RelTool(ReferencePoint,33,69,7\Rx:=19\Ry:=24\Rz:=0),velocity_edge,zone_edge,tool_nozzle\WObj:=wobj_substrate;
        MoveL RelTool(ReferencePoint,31,67,7\Rx:=24\Ry:=18\Rz:=0),velocity_edge,zone_edge,tool_nozzle\WObj:=wobj_substrate;
        MoveL RelTool(ReferencePoint,30,66,7\Rx:=27\Ry:=14\Rz:=0),velocity_edge,zone_edge,tool_nozzle\WObj:=wobj_substrate;
        MoveL RelTool(ReferencePoint,28,65,7\Rx:=29\Ry:=7\Rz:=0),velocity_edge,zone_edge,tool_nozzle\WObj:=wobj_substrate;
        MoveL RelTool(ReferencePoint,26,65,7\Rx:=30\Ry:=3\Rz:=0),velocity_edge,zone_edge,tool_nozzle\WObj:=wobj_substrate;
        MoveL RelTool(ReferencePoint,24,65,7\Rx:=30\Ry:=-4\Rz:=0),velocity_edge,zone_edge,tool_nozzle\WObj:=wobj_substrate;
        MoveL RelTool(ReferencePoint,22,66,7\Rx:=29\Ry:=-9\Rz:=0),velocity_edge,zone_edge,tool_nozzle\WObj:=wobj_substrate;
        MoveL RelTool(ReferencePoint,20,66,7\Rx:=26\Ry:=-15\Rz:=0),velocity_edge,zone_edge,tool_nozzle\WObj:=wobj_substrate;
        MoveL RelTool(ReferencePoint,18,67,7\Rx:=23\Ry:=-20\Rz:=0),velocity_edge,zone_edge,tool_nozzle\WObj:=wobj_substrate;
        MoveL RelTool(ReferencePoint,17,69,7\Rx:=19\Ry:=-24\Rz:=0),velocity_edge,zone_edge,tool_nozzle\WObj:=wobj_substrate;
        MoveL RelTool(ReferencePoint,16,71,7\Rx:=14\Ry:=-27\Rz:=0),velocity_edge,zone_edge,tool_nozzle\WObj:=wobj_substrate;
        MoveL RelTool(ReferencePoint,15,72,7\Rx:=9\Ry:=-29\Rz:=0),velocity_edge,zone_edge,tool_nozzle\WObj:=wobj_substrate;
        MoveL RelTool(ReferencePoint,15,74,7\Rx:=2\Ry:=-30\Rz:=0),velocity_edge,zone_edge,tool_nozzle\WObj:=wobj_substrate;
        MoveL RelTool(ReferencePoint,15,76,7\Rx:=-5\Ry:=-30\Rz:=0),velocity_edge,zone_edge,tool_nozzle\WObj:=wobj_substrate;
        MoveL RelTool(ReferencePoint,16,78,7\Rx:=-11\Ry:=-28\Rz:=0),velocity_edge,zone_edge,tool_nozzle\WObj:=wobj_substrate;
        MoveL RelTool(ReferencePoint,16,80,7\Rx:=-17\Ry:=-25\Rz:=0),velocity_edge,zone_edge,tool_nozzle\WObj:=wobj_substrate;
        MoveL RelTool(ReferencePoint,18,82,7\Rx:=-21\Ry:=-22\Rz:=0),velocity_edge,zone_edge,tool_nozzle\WObj:=wobj_substrate;
        MoveL RelTool(ReferencePoint,19,83,7\Rx:=-26\Ry:=-16\Rz:=0),velocity_edge,zone_edge,tool_nozzle\WObj:=wobj_substrate;
        MoveL RelTool(ReferencePoint,21,84,7\Rx:=-28\Ry:=-12\Rz:=0),velocity_edge,zone_edge,tool_nozzle\WObj:=wobj_substrate;
        MoveL RelTool(ReferencePoint,23,85,7\Rx:=-29\Ry:=-7\Rz:=0),velocity_edge,zone_edge,tool_nozzle\WObj:=wobj_substrate;
        MoveL RelTool(ReferencePoint,25,85,7\Rx:=-30\Ry:=-1\Rz:=0),velocity_edge,zone_edge,tool_nozzle\WObj:=wobj_substrate;
        MoveL RelTool(ReferencePoint,27,85,7\Rx:=-30\Ry:=4\Rz:=0),velocity_edge,zone_edge,tool_nozzle\WObj:=wobj_substrate;
        MoveL RelTool(ReferencePoint,28,85,7\Rx:=-29\Ry:=7\Rz:=0),velocity_edge,zone_edge,tool_nozzle\WObj:=wobj_substrate;
        MoveL RelTool(ReferencePoint,29,85,7\Rx:=0\Ry:=0\Rz:=0),velocity_link,zone_link,tool_nozzle\WObj:=wobj_substrate;
        MoveL RelTool(ReferencePoint,35,85,7\Rx:=0\Ry:=0\Rz:=0),velocity_link,zone_link,tool_nozzle\WObj:=wobj_substrate;
        MoveL RelTool(ReferencePoint,41,79,7\Rx:=0\Ry:=0\Rz:=0),velocity_link,zone_link,tool_nozzle\WObj:=wobj_substrate;
        MoveL RelTool(ReferencePoint,43,79,7\Rx:=0\Ry:=0\Rz:=0),velocity_link,zone_link,tool_nozzle\WObj:=wobj_substrate;
        MoveL RelTool(ReferencePoint,47,75,7\Rx:=0\Ry:=0\Rz:=0),velocity_link,zone_link,tool_nozzle\WObj:=wobj_substrate;
        MoveL RelTool(ReferencePoint,49,75,7\Rx:=0\Ry:=0\Rz:=0),velocity_link,zone_link,tool_nozzle\WObj:=wobj_substrate;
        MoveL RelTool(ReferencePoint,51,73,7\Rx:=0\Ry:=0\Rz:=0),velocity_link,zone_link,tool_nozzle\WObj:=wobj_substrate;
        MoveL RelTool(ReferencePoint,53,73,7\Rx:=0\Ry:=0\Rz:=0),velocity_link,zone_link,tool_nozzle\WObj:=wobj_substrate;
        MoveL RelTool(ReferencePoint,55,71,7\Rx:=0\Ry:=0\Rz:=0),velocity_link,zone_link,tool_nozzle\WObj:=wobj_substrate;
        MoveL RelTool(ReferencePoint,57,71,7\Rx:=0\Ry:=0\Rz:=0),velocity_link,zone_link,tool_nozzle\WObj:=wobj_substrate;
        MoveL RelTool(ReferencePoint,59,69,7\Rx:=0\Ry:=0\Rz:=0),velocity_link,zone_link,tool_nozzle\WObj:=wobj_substrate;
        MoveL RelTool(ReferencePoint,67,69,7\Rx:=0\Ry:=0\Rz:=0),velocity_link,zone_link,tool_nozzle\WObj:=wobj_substrate;
        MoveL RelTool(ReferencePoint,67,67,7\Rx:=0\Ry:=0\Rz:=0),velocity_infill,zone_infill,tool_nozzle\WObj:=wobj_substrate;
        MoveL RelTool(ReferencePoint,67,67,7\Rx:=0\Ry:=0\Rz:=0),velocity_infill,zone_infill,tool_nozzle\WObj:=wobj_substrate;
        MoveL RelTool(ReferencePoint,70,67,7\Rx:=0\Ry:=0\Rz:=0),velocity_infill,zone_infill,tool_nozzle\WObj:=wobj_substrate;
        MoveL RelTool(ReferencePoint,67,70,7\Rx:=0\Ry:=0\Rz:=0),velocity_infill,zone_infill,tool_nozzle\WObj:=wobj_substrate;
        MoveL RelTool(ReferencePoint,67,73,7\Rx:=0\Ry:=0\Rz:=0),velocity_infill,zone_infill,tool_nozzle\WObj:=wobj_substrate;
        MoveL RelTool(ReferencePoint,73,67,7\Rx:=0\Ry:=0\Rz:=0),velocity_infill,zone_infill,tool_nozzle\WObj:=wobj_substrate;
        MoveL RelTool(ReferencePoint,76,67,7\Rx:=0\Ry:=0\Rz:=0),velocity_infill,zone_infill,tool_nozzle\WObj:=wobj_substrate;
        MoveL RelTool(ReferencePoint,67,76,7\Rx:=0\Ry:=0\Rz:=0),velocity_infill,zone_infill,tool_nozzle\WObj:=wobj_substrate;
        MoveL RelTool(ReferencePoint,67,79,7\Rx:=0\Ry:=0\Rz:=0),velocity_infill,zone_infill,tool_nozzle\WObj:=wobj_substrate;
        MoveL RelTool(ReferencePoint,79,67,7\Rx:=0\Ry:=0\Rz:=0),velocity_infill,zone_infill,tool_nozzle\WObj:=wobj_substrate;
        MoveL RelTool(ReferencePoint,82,67,7\Rx:=0\Ry:=0\Rz:=0),velocity_infill,zone_infill,tool_nozzle\WObj:=wobj_substrate;
        MoveL RelTool(ReferencePoint,67,82,7\Rx:=0\Ry:=0\Rz:=0),velocity_infill,zone_infill,tool_nozzle\WObj:=wobj_substrate;
        MoveL RelTool(ReferencePoint,68,83,7\Rx:=0\Ry:=0\Rz:=0),velocity_infill,zone_infill,tool_nozzle\WObj:=wobj_substrate;
        MoveL RelTool(ReferencePoint,83,68,7\Rx:=0\Ry:=0\Rz:=0),velocity_infill,zone_infill,tool_nozzle\WObj:=wobj_substrate;
        MoveL RelTool(ReferencePoint,83,71,7\Rx:=0\Ry:=0\Rz:=0),velocity_infill,zone_infill,tool_nozzle\WObj:=wobj_substrate;
        MoveL RelTool(ReferencePoint,71,83,7\Rx:=0\Ry:=0\Rz:=0),velocity_infill,zone_infill,tool_nozzle\WObj:=wobj_substrate;
        MoveL RelTool(ReferencePoint,74,83,7\Rx:=0\Ry:=0\Rz:=0),velocity_infill,zone_infill,tool_nozzle\WObj:=wobj_substrate;
        MoveL RelTool(ReferencePoint,83,74,7\Rx:=0\Ry:=0\Rz:=0),velocity_infill,zone_infill,tool_nozzle\WObj:=wobj_substrate;
        MoveL RelTool(ReferencePoint,83,77,7\Rx:=0\Ry:=0\Rz:=0),velocity_infill,zone_infill,tool_nozzle\WObj:=wobj_substrate;
        MoveL RelTool(ReferencePoint,77,83,7\Rx:=0\Ry:=0\Rz:=0),velocity_infill,zone_infill,tool_nozzle\WObj:=wobj_substrate;
        MoveL RelTool(ReferencePoint,80,83,7\Rx:=0\Ry:=0\Rz:=0),velocity_infill,zone_infill,tool_nozzle\WObj:=wobj_substrate;
        MoveL RelTool(ReferencePoint,83,80,7\Rx:=0\Ry:=0\Rz:=0),velocity_infill,zone_infill,tool_nozzle\WObj:=wobj_substrate;
        MoveL RelTool(ReferencePoint,83,83,7\Rx:=0\Ry:=0\Rz:=0),velocity_infill,zone_infill,tool_nozzle\WObj:=wobj_substrate;
        MoveL RelTool(ReferencePoint,83,83,7\Rx:=0\Ry:=0\Rz:=0),velocity_infill,zone_infill,tool_nozzle\WObj:=wobj_substrate;
        MoveL RelTool(ReferencePoint,85,85,7\Rx:=0\Ry:=30\Rz:=0),velocity_edge,zone_edge,tool_nozzle\WObj:=wobj_substrate;
        MoveL RelTool(ReferencePoint,85,83,7\Rx:=0\Ry:=30\Rz:=0),velocity_edge,zone_edge,tool_nozzle\WObj:=wobj_substrate;
        MoveL RelTool(ReferencePoint,85,81,7\Rx:=0\Ry:=30\Rz:=0),velocity_edge,zone_edge,tool_nozzle\WObj:=wobj_substrate;
        MoveL RelTool(ReferencePoint,85,79,7\Rx:=0\Ry:=30\Rz:=0),velocity_edge,zone_edge,tool_nozzle\WObj:=wobj_substrate;
        MoveL RelTool(ReferencePoint,85,77,7\Rx:=0\Ry:=30\Rz:=0),velocity_edge,zone_edge,tool_nozzle\WObj:=wobj_substrate;
        MoveL RelTool(ReferencePoint,85,75,7\Rx:=0\Ry:=30\Rz:=0),velocity_edge,zone_edge,tool_nozzle\WObj:=wobj_substrate;
        MoveL RelTool(ReferencePoint,85,73,7\Rx:=0\Ry:=30\Rz:=0),velocity_edge,zone_edge,tool_nozzle\WObj:=wobj_substrate;
        MoveL RelTool(ReferencePoint,85,71,7\Rx:=0\Ry:=30\Rz:=0),velocity_edge,zone_edge,tool_nozzle\WObj:=wobj_substrate;
        MoveL RelTool(ReferencePoint,85,69,7\Rx:=0\Ry:=30\Rz:=0),velocity_edge,zone_edge,tool_nozzle\WObj:=wobj_substrate;
        MoveL RelTool(ReferencePoint,85,67,7\Rx:=0\Ry:=30\Rz:=0),velocity_edge,zone_edge,tool_nozzle\WObj:=wobj_substrate;
        MoveL RelTool(ReferencePoint,85,65,7\Rx:=30\Ry:=0\Rz:=0),velocity_edge,zone_edge,tool_nozzle\WObj:=wobj_substrate;
        MoveL RelTool(ReferencePoint,83,65,7\Rx:=30\Ry:=0\Rz:=0),velocity_edge,zone_edge,tool_nozzle\WObj:=wobj_substrate;
        MoveL RelTool(ReferencePoint,81,65,7\Rx:=30\Ry:=0\Rz:=0),velocity_edge,zone_edge,tool_nozzle\WObj:=wobj_substrate;
        MoveL RelTool(ReferencePoint,79,65,7\Rx:=30\Ry:=0\Rz:=0),velocity_edge,zone_edge,tool_nozzle\WObj:=wobj_substrate;
        MoveL RelTool(ReferencePoint,77,65,7\Rx:=30\Ry:=0\Rz:=0),velocity_edge,zone_edge,tool_nozzle\WObj:=wobj_substrate;
        MoveL RelTool(ReferencePoint,75,65,7\Rx:=30\Ry:=0\Rz:=0),velocity_edge,zone_edge,tool_nozzle\WObj:=wobj_substrate;
        MoveL RelTool(ReferencePoint,73,65,7\Rx:=30\Ry:=0\Rz:=0),velocity_edge,zone_edge,tool_nozzle\WObj:=wobj_substrate;
        MoveL RelTool(ReferencePoint,71,65,7\Rx:=30\Ry:=0\Rz:=0),velocity_edge,zone_edge,tool_nozzle\WObj:=wobj_substrate;
        MoveL RelTool(ReferencePoint,69,65,7\Rx:=30\Ry:=0\Rz:=0),velocity_edge,zone_edge,tool_nozzle\WObj:=wobj_substrate;
        MoveL RelTool(ReferencePoint,67,65,7\Rx:=30\Ry:=0\Rz:=0),velocity_edge,zone_edge,tool_nozzle\WObj:=wobj_substrate;
        MoveL RelTool(ReferencePoint,65,65,7\Rx:=0\Ry:=-30\Rz:=0),velocity_edge,zone_edge,tool_nozzle\WObj:=wobj_substrate;
        MoveL RelTool(ReferencePoint,65,67,7\Rx:=0\Ry:=-30\Rz:=0),velocity_edge,zone_edge,tool_nozzle\WObj:=wobj_substrate;
        MoveL RelTool(ReferencePoint,65,69,7\Rx:=0\Ry:=-30\Rz:=0),velocity_edge,zone_edge,tool_nozzle\WObj:=wobj_substrate;
        MoveL RelTool(ReferencePoint,65,71,7\Rx:=0\Ry:=-30\Rz:=0),velocity_edge,zone_edge,tool_nozzle\WObj:=wobj_substrate;
        MoveL RelTool(ReferencePoint,65,73,7\Rx:=0\Ry:=-30\Rz:=0),velocity_edge,zone_edge,tool_nozzle\WObj:=wobj_substrate;
        MoveL RelTool(ReferencePoint,65,75,7\Rx:=0\Ry:=-30\Rz:=0),velocity_edge,zone_edge,tool_nozzle\WObj:=wobj_substrate;
        MoveL RelTool(ReferencePoint,65,77,7\Rx:=0\Ry:=-30\Rz:=0),velocity_edge,zone_edge,tool_nozzle\WObj:=wobj_substrate;
        MoveL RelTool(ReferencePoint,65,79,7\Rx:=0\Ry:=-30\Rz:=0),velocity_edge,zone_edge,tool_nozzle\WObj:=wobj_substrate;
        MoveL RelTool(ReferencePoint,65,81,7\Rx:=0\Ry:=-30\Rz:=0),velocity_edge,zone_edge,tool_nozzle\WObj:=wobj_substrate;
        MoveL RelTool(ReferencePoint,65,83,7\Rx:=0\Ry:=-30\Rz:=0),velocity_edge,zone_edge,tool_nozzle\WObj:=wobj_substrate;
        MoveL RelTool(ReferencePoint,65,85,7\Rx:=-30\Ry:=0\Rz:=0),velocity_edge,zone_edge,tool_nozzle\WObj:=wobj_substrate;
        MoveL RelTool(ReferencePoint,67,85,7\Rx:=-30\Ry:=0\Rz:=0),velocity_edge,zone_edge,tool_nozzle\WObj:=wobj_substrate;
        MoveL RelTool(ReferencePoint,69,85,7\Rx:=-30\Ry:=0\Rz:=0),velocity_edge,zone_edge,tool_nozzle\WObj:=wobj_substrate;
        MoveL RelTool(ReferencePoint,71,85,7\Rx:=-30\Ry:=0\Rz:=0),velocity_edge,zone_edge,tool_nozzle\WObj:=wobj_substrate;
        MoveL RelTool(ReferencePoint,73,85,7\Rx:=-30\Ry:=0\Rz:=0),velocity_edge,zone_edge,tool_nozzle\WObj:=wobj_substrate;
        MoveL RelTool(ReferencePoint,75,85,7\Rx:=-30\Ry:=0\Rz:=0),velocity_edge,zone_edge,tool_nozzle\WObj:=wobj_substrate;
        MoveL RelTool(ReferencePoint,77,85,7\Rx:=-30\Ry:=0\Rz:=0),velocity_edge,zone_edge,tool_nozzle\WObj:=wobj_substrate;
        MoveL RelTool(ReferencePoint,79,85,7\Rx:=-30\Ry:=0\Rz:=0),velocity_edge,zone_edge,tool_nozzle\WObj:=wobj_substrate;
        MoveL RelTool(ReferencePoint,81,85,7\Rx:=-30\Ry:=0\Rz:=0),velocity_edge,zone_edge,tool_nozzle\WObj:=wobj_substrate;
        MoveL RelTool(ReferencePoint,83,85,7\Rx:=-30\Ry:=0\Rz:=0),velocity_edge,zone_edge,tool_nozzle\WObj:=wobj_substrate;
        MoveL RelTool(ReferencePoint,85,85,7\Rx:=-30\Ry:=0\Rz:=0),velocity_edge,zone_edge,tool_nozzle\WObj:=wobj_substrate;
        MoveL Offs(StartPoint,0,0,27),v100,fine,tool_nozzle\WObj:=wobj_substrate;
    ENDPROC
ENDMODULE
